// TwinCAT 3 PLC project
// project tree:
//   POUs/ makeTupleStruct_1.TcPOU, proj0_TupleStruct_1.TcPOU, proj1_TupleStruct_1.TcPOU, proj2_TupleStruct_1.TcPOU, proj3_TupleStruct_1.TcPOU, proj4_TupleStruct_1.TcPOU, proj5_TupleStruct_1.TcPOU, proj6_TupleStruct_1.TcPOU, proj7_TupleStruct_1.TcPOU, proj8_TupleStruct_1.TcPOU, proj9_TupleStruct_1.TcPOU, proj10_TupleStruct_1.TcPOU, proj11_TupleStruct_1.TcPOU, proj12_TupleStruct_1.TcPOU, proj13_TupleStruct_1.TcPOU, MAIN.TcPOU
//   DUTs/ STATE.TcDUT, enum_E.TcDUT, TupleStruct_1.TcDUT
//   GVLs/ TIMERS.TcGVL (not stored)

// ---- DUTs/STATE.TcDUT
TYPE STATE:
    STRUCT
        curTime: LREAL;
        dvar_M_p_v0 AT %Q*: LREAL;
        dvar_M_p_v1 AT %Q*: DINT;
        dvar_M_p_v2 AT %Q*: DINT;
        dvar_M_p_v3 AT %Q*: DINT;
        dvar_M_p_v99 AT %Q*: LREAL;
        dvar_M_p_vx AT %Q*: LREAL;
        dvar_M_p_vr AT %Q*: TupleStruct_1;
        dvar_M_p AT %Q*: enum_E;
    END_STRUCT
END_TYPE

// ---- DUTs/enum_E.TcDUT
TYPE enum_E:
    (elit_m1, elit_m2);
END_TYPE

// ---- DUTs/TupleStruct_1.TcDUT

      TYPE TupleStruct_1:
    STRUCT
        field0: LREAL;
        field1: LREAL;
        field2: LREAL;
        field3: LREAL;
        field4: LREAL;
        field5: LREAL;
        field6: LREAL;
        field7: LREAL;
        field8: LREAL;
        field9: LREAL;
        field10: LREAL;
        field11: LREAL;
        field12: LREAL;
        field13: LREAL;
    END_STRUCT
END_TYPE

// ---- POUs/makeTupleStruct_1.TcPOU

      FUNCTION makeTupleStruct_1: TupleStruct_1
VAR_INPUT
    field0: LREAL;
    field1: LREAL;
    field2: LREAL;
    field3: LREAL;
    field4: LREAL;
    field5: LREAL;
    field6: LREAL;
    field7: LREAL;
    field8: LREAL;
    field9: LREAL;
    field10: LREAL;
    field11: LREAL;
    field12: LREAL;
    field13: LREAL;
END_VAR
VAR
    rslt: TupleStruct_1;
END_VAR


        rslt.field0 := field0;
rslt.field1 := field1;
rslt.field2 := field2;
rslt.field3 := field3;
rslt.field4 := field4;
rslt.field5 := field5;
rslt.field6 := field6;
rslt.field7 := field7;
rslt.field8 := field8;
rslt.field9 := field9;
rslt.field10 := field10;
rslt.field11 := field11;
rslt.field12 := field12;
rslt.field13 := field13;
makeTupleStruct_1 := rslt;

END_FUNCTION

// ---- POUs/proj0_TupleStruct_1.TcPOU
FUNCTION proj0_TupleStruct_1: LREAL
VAR_INPUT
    tuple: TupleStruct_1;
END_VAR

proj0_TupleStruct_1 := tuple.field0;

END_FUNCTION

// ---- POUs/proj1_TupleStruct_1.TcPOU
FUNCTION proj1_TupleStruct_1: LREAL
VAR_INPUT
    tuple: TupleStruct_1;
END_VAR

proj1_TupleStruct_1 := tuple.field1;

END_FUNCTION

// ---- POUs/proj2_TupleStruct_1.TcPOU
FUNCTION proj2_TupleStruct_1: LREAL
VAR_INPUT
    tuple: TupleStruct_1;
END_VAR

proj2_TupleStruct_1 := tuple.field2;

END_FUNCTION

// ---- POUs/proj3_TupleStruct_1.TcPOU

      FUNCTION proj3_TupleStruct_1: LREAL
VAR_INPUT
    tuple: TupleStruct_1;
END_VAR


        proj3_TupleStruct_1 := tuple.field3;

END_FUNCTION

// ---- POUs/proj4_TupleStruct_1.TcPOU

      FUNCTION proj4_TupleStruct_1: LREAL
VAR_INPUT
    tuple: TupleStruct_1;
END_VAR


        proj4_TupleStruct_1 := tuple.field4;

END_FUNCTION

// ---- POUs/proj5_TupleStruct_1.TcPOU
FUNCTION proj5_TupleStruct_1: LREAL
VAR_INPUT
    tuple: TupleStruct_1;
END_VAR

proj5_TupleStruct_1 := tuple.field5;

END_FUNCTION

// ---- POUs/proj6_TupleStruct_1.TcPOU

      FUNCTION proj6_TupleStruct_1: LREAL
VAR_INPUT
    tuple: TupleStruct_1;
END_VAR


        proj6_TupleStruct_1 := tuple.field6;

END_FUNCTION

// ---- POUs/proj7_TupleStruct_1.TcPOU
FUNCTION proj7_TupleStruct_1: LREAL
VAR_INPUT
    tuple: TupleStruct_1;
END_VAR

proj7_TupleStruct_1 := tuple.field7;

END_FUNCTION

// ---- POUs/proj8_TupleStruct_1.TcPOU

      FUNCTION proj8_TupleStruct_1: LREAL
VAR_INPUT
    tuple: TupleStruct_1;
END_VAR


        proj8_TupleStruct_1 := tuple.field8;

END_FUNCTION

// ---- POUs/proj9_TupleStruct_1.TcPOU
FUNCTION proj9_TupleStruct_1: LREAL
VAR_INPUT
    tuple: TupleStruct_1;
END_VAR

proj9_TupleStruct_1 := tuple.field9;

END_FUNCTION

// ---- POUs/proj10_TupleStruct_1.TcPOU

      FUNCTION proj10_TupleStruct_1: LREAL
VAR_INPUT
    tuple: TupleStruct_1;
END_VAR


        proj10_TupleStruct_1 := tuple.field10;

END_FUNCTION

// ---- POUs/proj11_TupleStruct_1.TcPOU

      FUNCTION proj11_TupleStruct_1: LREAL
VAR_INPUT
    tuple: TupleStruct_1;
END_VAR


        proj11_TupleStruct_1 := tuple.field11;

END_FUNCTION

// ---- POUs/proj12_TupleStruct_1.TcPOU
FUNCTION proj12_TupleStruct_1: LREAL
VAR_INPUT
    tuple: TupleStruct_1;
END_VAR

proj12_TupleStruct_1 := tuple.field12;

END_FUNCTION

// ---- POUs/proj13_TupleStruct_1.TcPOU
FUNCTION proj13_TupleStruct_1: LREAL
VAR_INPUT
    tuple: TupleStruct_1;
END_VAR

proj13_TupleStruct_1 := tuple.field13;

END_FUNCTION

// ---- POUs/MAIN.TcPOU

      PROGRAM MAIN
VAR_OUTPUT
    timerValue0: TIME;
    timerValue1: TIME;
END_VAR
VAR
    cnt: LINT;
    first: BOOL := TRUE;
    curTimerValue: TIME;
    state0: STATE;
    curTime: LREAL;
    loopsKilled: LINT;
END_VAR
VAR_TEMP
    lastTimerValue: TIME;
    curDeltaTime: TIME;
    curDeltaSecs: LREAL;
    state1: STATE;
    progress: BOOL;
    loopCount: INT;
END_VAR


        
// Handle 'time' and cycle time.
cnt := cnt + 1;

timer0(IN := curTimer = 0, PT := T#1D);
timer1(IN := curTimer = 1, PT := T#1D);
timerValue0 := timer0.ET;
timerValue1 := timer1.ET;

lastTimerValue := curTimerValue;
IF curTimer = 0 THEN
    curTimerValue := timerValue0;
ELSE
    curTimerValue := timerValue1;
END_IF;
curDeltaTime := curTimerValue - lastTimerValue;
curDeltaSecs := TIME_TO_LREAL(curDeltaTime) / 1000;
curTime := curTime + curDeltaSecs;

IF cnt MOD 10 = 0 THEN
    curTimer := 1 - curTimer;
    curTimerValue := T#0S;
    timer0(IN := curTimer = 0, PT := T#1D);
    timer1(IN := curTimer = 1, PT := T#1D);
    timerValue0 := timer0.ET;
    timerValue1 := timer1.ET;
END_IF;

IF first THEN
    first := FALSE;

    // Initialize state variables for initial state.
    state0.dvar_M_p_v0 := 0.0;
    state0.dvar_M_p_v1 := 1;
    state0.dvar_M_p_v2 := 2;
    state0.dvar_M_p_v3 := 3;
    state0.dvar_M_p_v99 := 1.0e99;
    state0.dvar_M_p_vx := 0.0;
    state0.dvar_M_p_vr := makeTupleStruct_1(1.0, 1.0, 1.0, 1.0, 1.0, 1.0, 1.0, 1.0, 1.0, 1.0, 1.0, 1.0, 1.0, 1.0);
    state0.dvar_M_p := elit_m1;
ELSE
    // Update continuous variables for time delay.

    state0.curTime := curTime;
END_IF;

// Event loop.
WHILE TRUE DO
    progress := FALSE;

    // Event "tau".
    IF NOT progress THEN
        IF (state0.dvar_M_p) = (elit_m1) THEN
            progress := TRUE;
            state1 := state0;

            state1.dvar_M_p_vr := makeTupleStruct_1(-(state0.dvar_M_p_v0), -(-(-(state0.dvar_M_p_v0))), -(-(-(-(-(state0.dvar_M_p_v0))))), (state0.dvar_M_p_v0) * (-1.0), (state0.dvar_M_p_v0) / (-1), (-4.9e-324) / (state0.dvar_M_p_v99), EXPT(-(state0.dvar_M_p_v0), 1.0/3), LN((state0.dvar_M_p_v1) - (1.0e-18)), LN((state0.dvar_M_p_v1) - (1.0e-17)), LN((state0.dvar_M_p_v1) - (1.0e-16)), EXPT(-1.0e-300, state0.dvar_M_p_v1), EXPT(-1.0e-300, state0.dvar_M_p_v2), EXPT(-1.0e-300, state0.dvar_M_p_v3), -(state0.dvar_M_p_vx));
            state1.dvar_M_p := elit_m2;

            state0 := state1;
        END_IF;
    END_IF;

    // Done with events?
    IF NOT progress THEN
        EXIT;
    END_IF;

    // Protect against events that are always enabled.
    loopCount := loopCount + 1;
    IF loopCount >= 100 THEN
        loopsKilled := loopsKilled + 1;
        EXIT;
    END_IF;
END_WHILE;

END_PROGRAM
